Staubli VAL3: consumeAny.pgx

program consumeAny(num& x_nStatus (dimensions=1))
  local num l_nData[4]
begin
  // consumes 4 bytes and verifes with the reference
  // does nothing if first return parameter is not 0
  // return
  //    -2 - timeout
  //    -1 - unsuccessful
  //     0 - successfuly received (consumed) 4 bytes
  if x_nStatus<0
    return
  endIf
  x_nStatus=sioGet(siConn,l_nData)
  if x_nStatus==4
    x_nStatus=0
  elseIf x_nStatus==-1
    x_nStatus=-2
  else
    x_nStatus=-1
  endIf
end
